{attribute 'GeneratedUsingTerminal: EJ1957-0000-0017'}
{attribute addProperty BoxType "EJ1957-0000-0017"}
{attribute addProperty Id "FSOEAT %Q*FSOE_D1C9D1EA14"}
{attribute addProperty CRC "524341507"}
{attribute addProperty Size "14"}
TYPE FSoE_Outputs_1F40D103 :
STRUCT
	{attribute addProperty Name "FSOE"}
	FSOE AT %Q* : FSOE_D1C9D1EA;
END_STRUCT
END_TYPE

(* stored: Version 1.2.0.0, ProductVersion 3.1.4024.9
   DUT FSoE_Outputs_1F40D103: Id {0140fb29-f4ff-4c48-9365-54f7e402debd} *)
